FUNCTION_BLOCK FB_Rechazador_SFC
VAR_INPUT
	
	//Tiempo
	Tcheck: TIME := T#1S;	
	
	// SFC-Flags
	SFCPause: BOOL;
	SFCReset: BOOL;
	
	//Indicadores de sincronizacion
	Ack: BOOL:= TRUE;
	Execute: BOOL;
	
	//Entradas
	
	Verificador_abajo: BOOL;

	
END_VAR
VAR_OUTPUT
	//indicadores de sincronizacion
	Done: BOOL;
	Ready: BOOL;

	//Salidas
	Rechazador_adelante: BOOL;
	
END_VAR
VAR
END_VAR

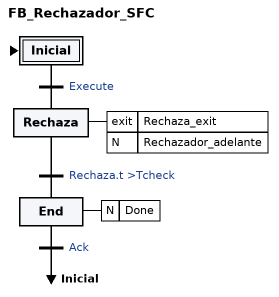
INITIAL_STEP Inicial:
END_STEP
TRANSITION FROM Inicial TO Rechaza
    := Execute;
END_TRANSITION
STEP Rechaza:
    Rechaza_exit(P0);  // exit action
    Rechazador_adelante(N);
END_STEP
TRANSITION FROM Rechaza TO End
    := Rechaza.t >Tcheck;
END_TRANSITION
STEP End:
    Done(N);
END_STEP
TRANSITION FROM End TO Inicial
    := Ack;
END_TRANSITION

ACTION Rechaza_exit:

END_ACTION

END_FUNCTION_BLOCK

(* stored: Version 1.1.0.1, ProductVersion 3.1.4024.12
   POU FB_Rechazador_SFC: Id {f4214f36-f1b2-4ea8-b61c-4ba01b83119c}, SpecialFunc None
   Action Rechaza_exit: Id {0d6b0c18-f0ed-4800-8a32-b185cb7b27ae} *)
